# EPICS substitutions: db/EL3162.substitutions
file EL3162.template
{ 	pattern
	{
		TERMINAL,
		DESC1,	SCAN1,	ADEL1,	EGUF1,	EGUL1,	HIGH1,	HIHI1,	HOPR1,	HYST1,	LOLO1,	LOPR1,	LOW1,	MDEL1,	SMOO1,	UNIT1,
		DESC2,	SCAN2,	ADEL2,	EGUF2,	EGUL2,	HIGH2,	HIHI2,	HOPR2,	HYST2,	LOLO2,	LOPR2,	LOW2,	MDEL2,	SMOO2,	UNIT2
	}
	{
	}
}
